// Mitsubishi GX Works2 project: 4LightsSeqLDv2   PLC: FX2N/FX2NC
// Examples Algorithm of 4 Lights on in seq then off in seq

// global labels: Global1
VAR_GLOBAL
  Step1 AT S10 : BOOL;  (* Inital Step *)
  Step2 AT S11 : BOOL;
  Step3 AT S12 : BOOL;
  Step4 AT S13 : BOOL;
  Step5 AT S14 : BOOL;
  Step6 AT S15 : BOOL;
  Step7 AT S16 : BOOL;
  Step8 AT S17 : BOOL;
  Step9 AT S18 : BOOL;
  StartPB AT X000 : BOOL;  (* NO Momentary PB *)
  StopPB AT X001 : BOOL;  (* NC Momentary PB *)
  PL1 AT Y000 : BOOL;
  PL2 AT Y001 : BOOL;
  PL3 AT Y002 : BOOL;
  PL4 AT Y003 : BOOL;
  SC : BOOL;  (* State Changed *)
  CurrentState AT D100 : WORD;
  PreviousState AT D101 : WORD;
  S1ToS2 : BOOL;
  S2ToS3 : BOOL;
  S3ToS4 : BOOL;
  S4ToS5 : BOOL;
  S5ToS6 : BOOL;
  S6ToS7 : BOOL;
  S7ToS8 : BOOL;
  S8ToS9 : BOOL;
  S9ToS1 : BOOL;
  Do_Shift : BOOL;
  Src_Bit : BOOL;
  First_Start : BOOL;
  Step0 AT S9 : BOOL;
  StepCtr : CTU;
  Stp_Ary : ARRAY [0..15] OF BOOL;
  Stp_Idx : INT;
  StpDn_Ary : ARRAY [0..15] OF BOOL;
  Get_Step_1 : Get_Step;
  Do_Count : BOOL;
  Stp_Ary_D : ARRAY [0..15] OF BOOL;
  StpDn_Ary_D : ARRAY [0..15] OF BOOL;
END_VAR

// task Task_01 (event TRUE, interval 0, priority 31): FSM_DRUM

PROGRAM FSM_SR_NO_SC
(* structured ladder/FBD written out as ST: instructions are called as NAME(EN, inputs, outputs); _pN, _eN, _tN stand for wires *)
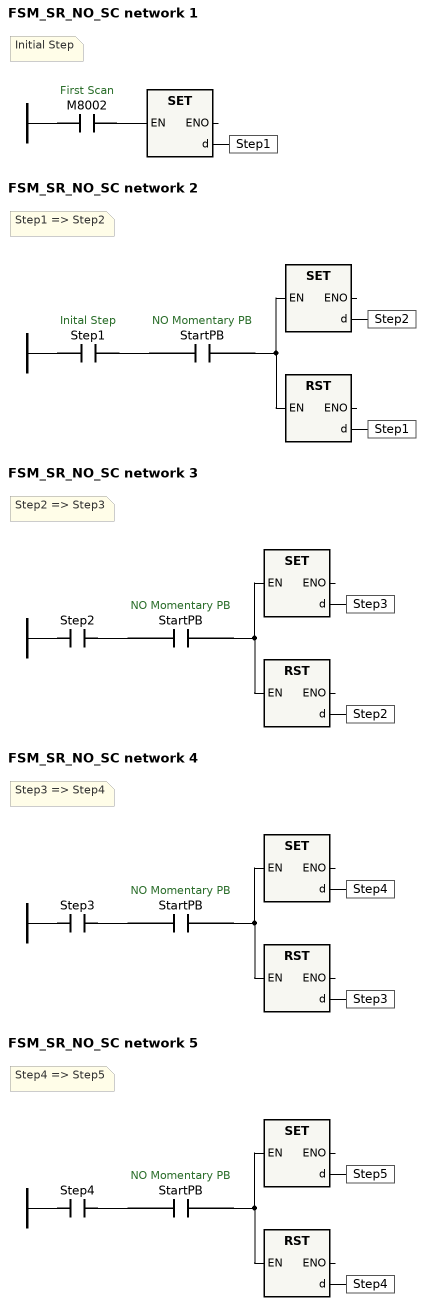
(* network 1 *)
(* Initial Step *)
SET(M8002, Step1);
(* network 2 *)
(* Step1 => Step2 *)
_p1 := Step1 AND StartPB;
SET(_p1, Step2);
RST(_p1, Step1);
(* network 3 *)
(* Step2 => Step3 *)
_p1 := Step2 AND StartPB;
SET(_p1, Step3);
RST(_p1, Step2);
(* network 4 *)
(* Step3 => Step4 *)
_p1 := Step3 AND StartPB;
SET(_p1, Step4);
RST(_p1, Step3);
(* network 5 *)
(* Step4 => Step5 *)
_p1 := Step4 AND StartPB;
SET(_p1, Step5);
RST(_p1, Step4);
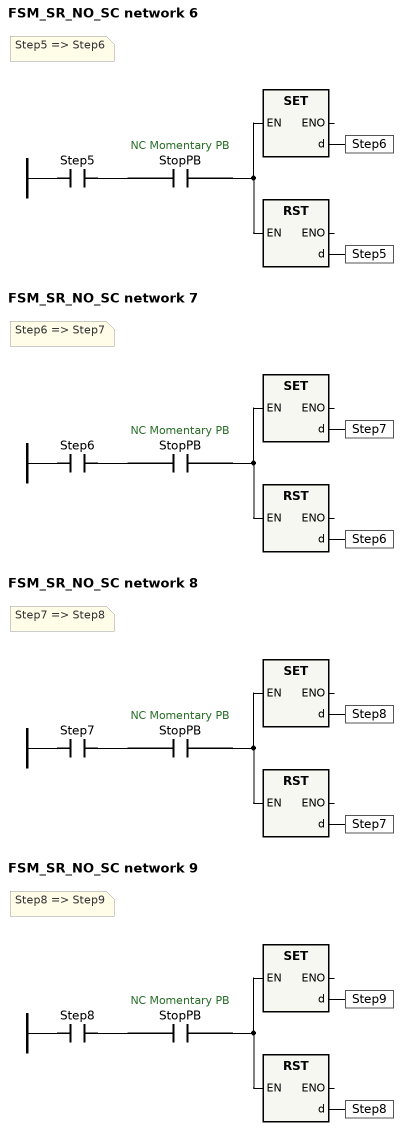
(* network 6 *)
(* Step5 => Step6 *)
_p1 := Step5 AND StopPB;
SET(_p1, Step6);
RST(_p1, Step5);
(* network 7 *)
(* Step6 => Step7 *)
_p1 := Step6 AND StopPB;
SET(_p1, Step7);
RST(_p1, Step6);
(* network 8 *)
(* Step7 => Step8 *)
_p1 := Step7 AND StopPB;
SET(_p1, Step8);
RST(_p1, Step7);
(* network 9 *)
(* Step8 => Step9 *)
_p1 := Step8 AND StopPB;
SET(_p1, Step9);
RST(_p1, Step8);
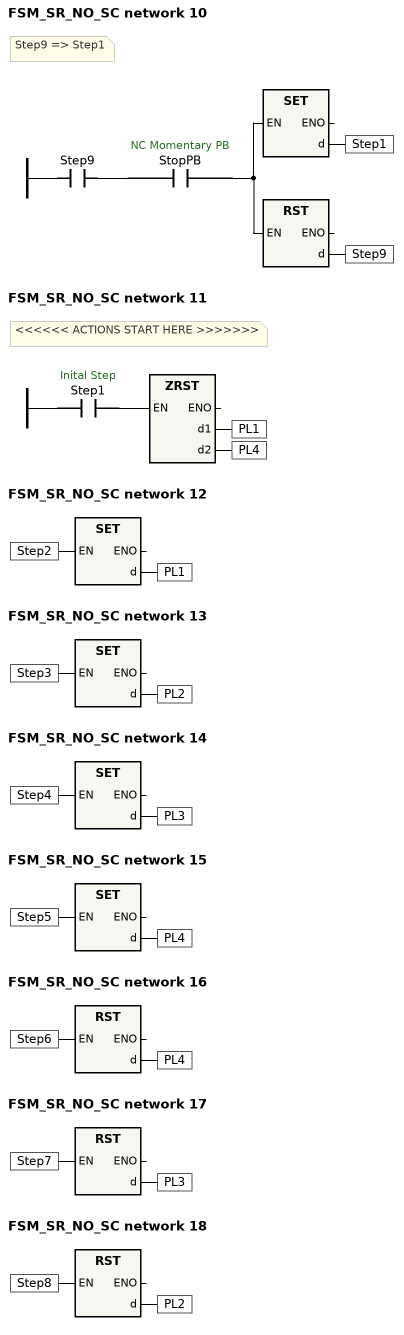
(* network 10 *)
(* Step9 => Step1 *)
_p1 := Step9 AND StopPB;
SET(_p1, Step1);
RST(_p1, Step9);
(* network 11 *)
(* <<<<<< ACTIONS START HERE >>>>>>> *)
ZRST(Step1, PL1, PL4);
(* network 12 *)
SET(Step2, PL1);
(* network 13 *)
SET(Step3, PL2);
(* network 14 *)
SET(Step4, PL3);
(* network 15 *)
SET(Step5, PL4);
(* network 16 *)
RST(Step6, PL4);
(* network 17 *)
RST(Step7, PL3);
(* network 18 *)
RST(Step8, PL2);
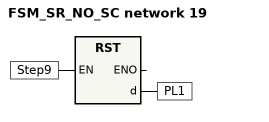
(* network 19 *)
RST(Step9, PL1);
END_PROGRAM

PROGRAM FSM_SR_SC
(* structured ladder/FBD written out as ST: instructions are called as NAME(EN, inputs, outputs); _pN, _eN, _tN stand for wires *)
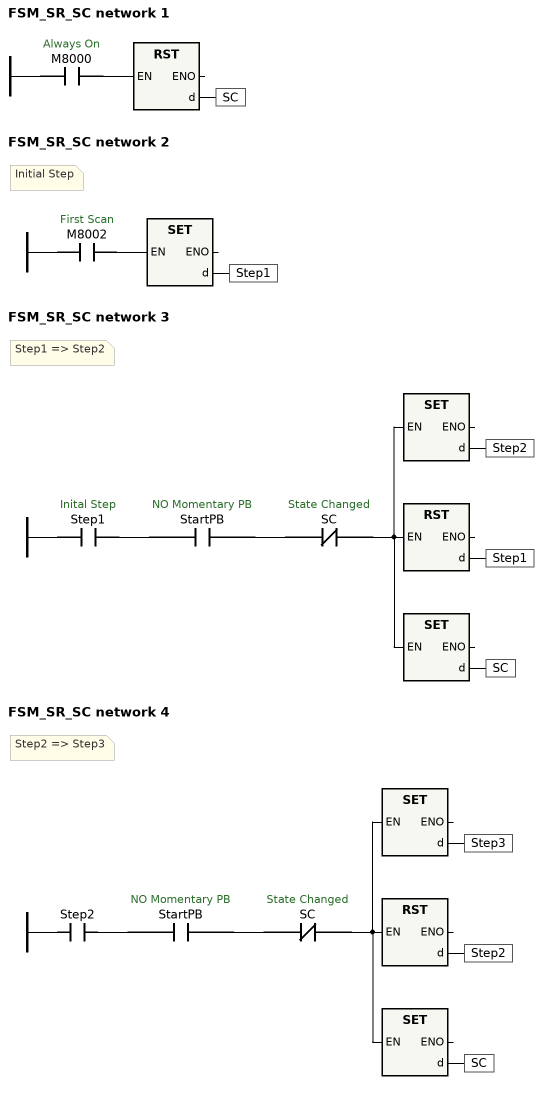
(* network 1 *)
RST(M8000, SC);
(* network 2 *)
(* Initial Step *)
SET(M8002, Step1);
(* network 3 *)
(* Step1 => Step2 *)
_p1 := Step1 AND StartPB AND NOT SC;
SET(_p1, Step2);
RST(_p1, Step1);
SET(_p1, SC);
(* network 4 *)
(* Step2 => Step3 *)
_p1 := Step2 AND StartPB AND NOT SC;
SET(_p1, Step3);
RST(_p1, Step2);
SET(_p1, SC);
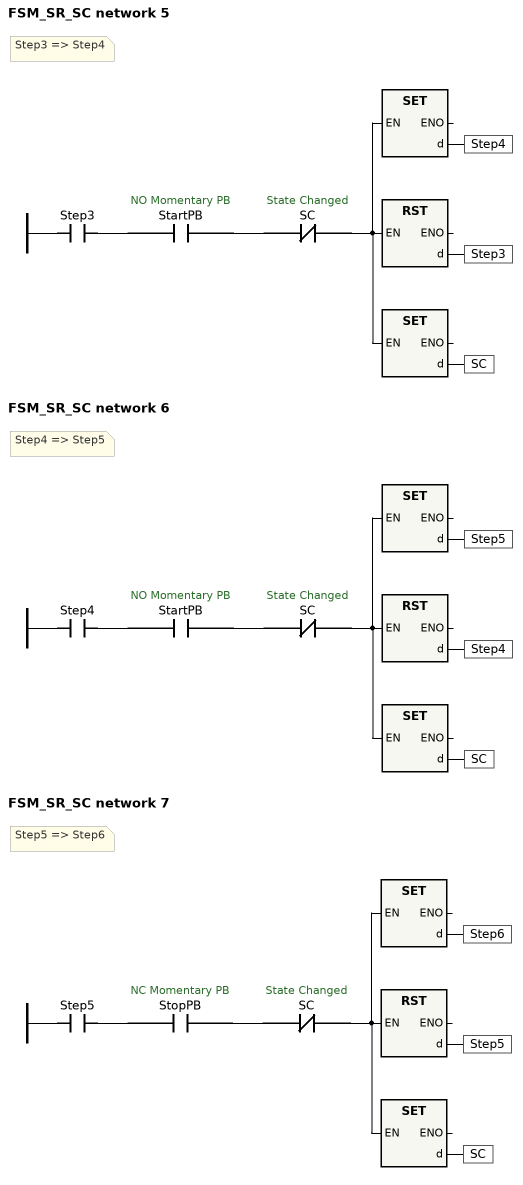
(* network 5 *)
(* Step3 => Step4 *)
_p1 := Step3 AND StartPB AND NOT SC;
SET(_p1, Step4);
RST(_p1, Step3);
SET(_p1, SC);
(* network 6 *)
(* Step4 => Step5 *)
_p1 := Step4 AND StartPB AND NOT SC;
SET(_p1, Step5);
RST(_p1, Step4);
SET(_p1, SC);
(* network 7 *)
(* Step5 => Step6 *)
_p1 := Step5 AND StopPB AND NOT SC;
SET(_p1, Step6);
RST(_p1, Step5);
SET(_p1, SC);
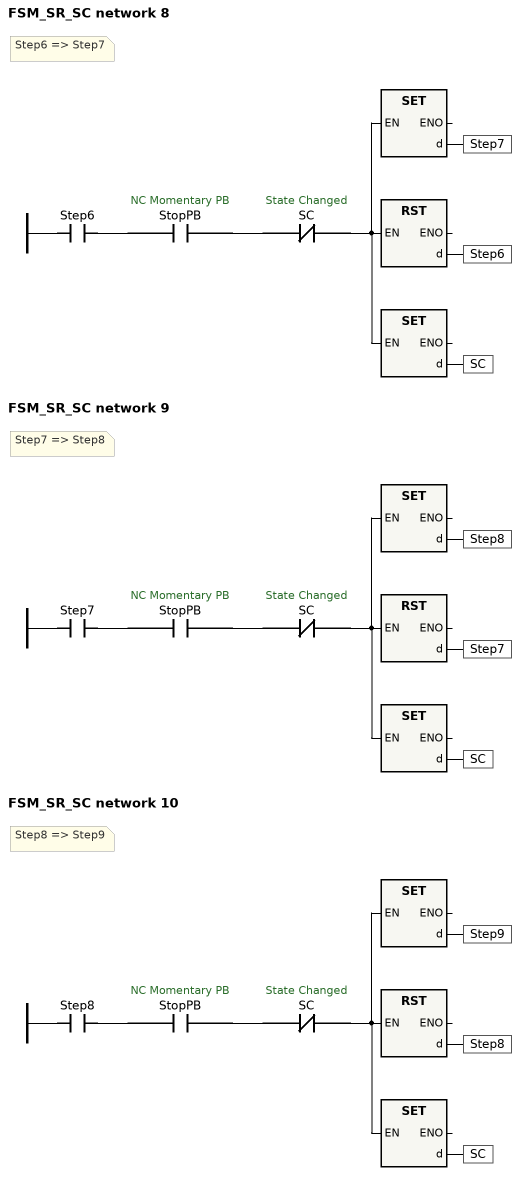
(* network 8 *)
(* Step6 => Step7 *)
_p1 := Step6 AND StopPB AND NOT SC;
SET(_p1, Step7);
RST(_p1, Step6);
SET(_p1, SC);
(* network 9 *)
(* Step7 => Step8 *)
_p1 := Step7 AND StopPB AND NOT SC;
SET(_p1, Step8);
RST(_p1, Step7);
SET(_p1, SC);
(* network 10 *)
(* Step8 => Step9 *)
_p1 := Step8 AND StopPB AND NOT SC;
SET(_p1, Step9);
RST(_p1, Step8);
SET(_p1, SC);
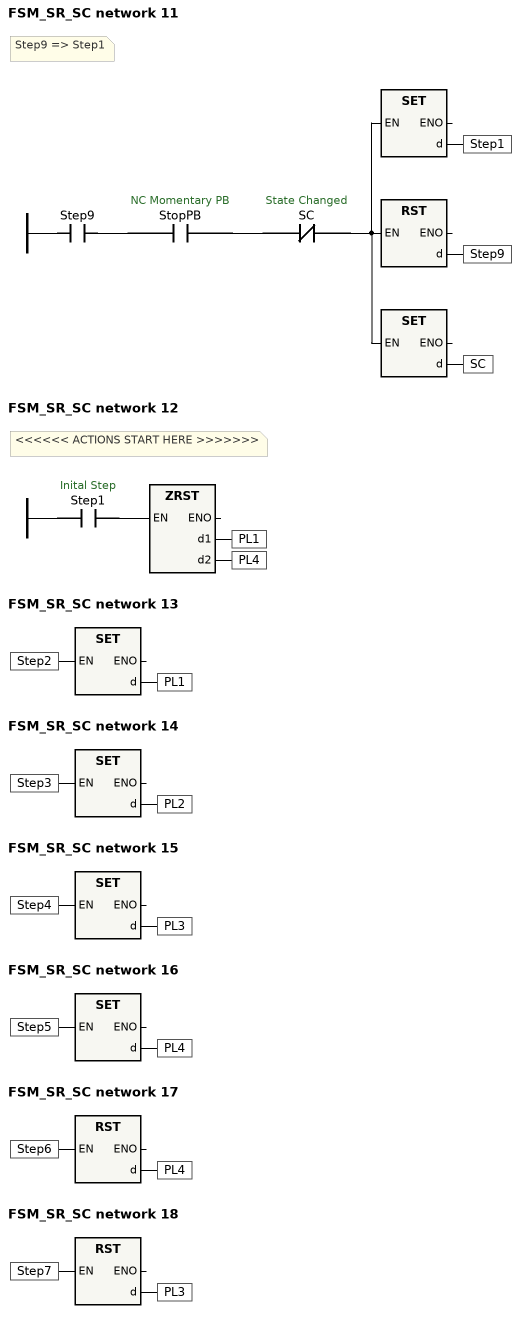
(* network 11 *)
(* Step9 => Step1 *)
_p1 := Step9 AND StopPB AND NOT SC;
SET(_p1, Step1);
RST(_p1, Step9);
SET(_p1, SC);
(* network 12 *)
(* <<<<<< ACTIONS START HERE >>>>>>> *)
ZRST(Step1, PL1, PL4);
(* network 13 *)
SET(Step2, PL1);
(* network 14 *)
SET(Step3, PL2);
(* network 15 *)
SET(Step4, PL3);
(* network 16 *)
SET(Step5, PL4);
(* network 17 *)
RST(Step6, PL4);
(* network 18 *)
RST(Step7, PL3);
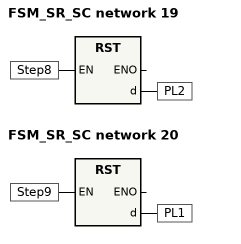
(* network 19 *)
RST(Step8, PL2);
(* network 20 *)
RST(Step9, PL1);
END_PROGRAM

PROGRAM FSM_EQU
(* structured ladder/FBD written out as ST: instructions are called as NAME(EN, inputs, outputs); _pN, _eN, _tN stand for wires *)
(* Instructions Supported in Simulator and LE3U Trainer *)
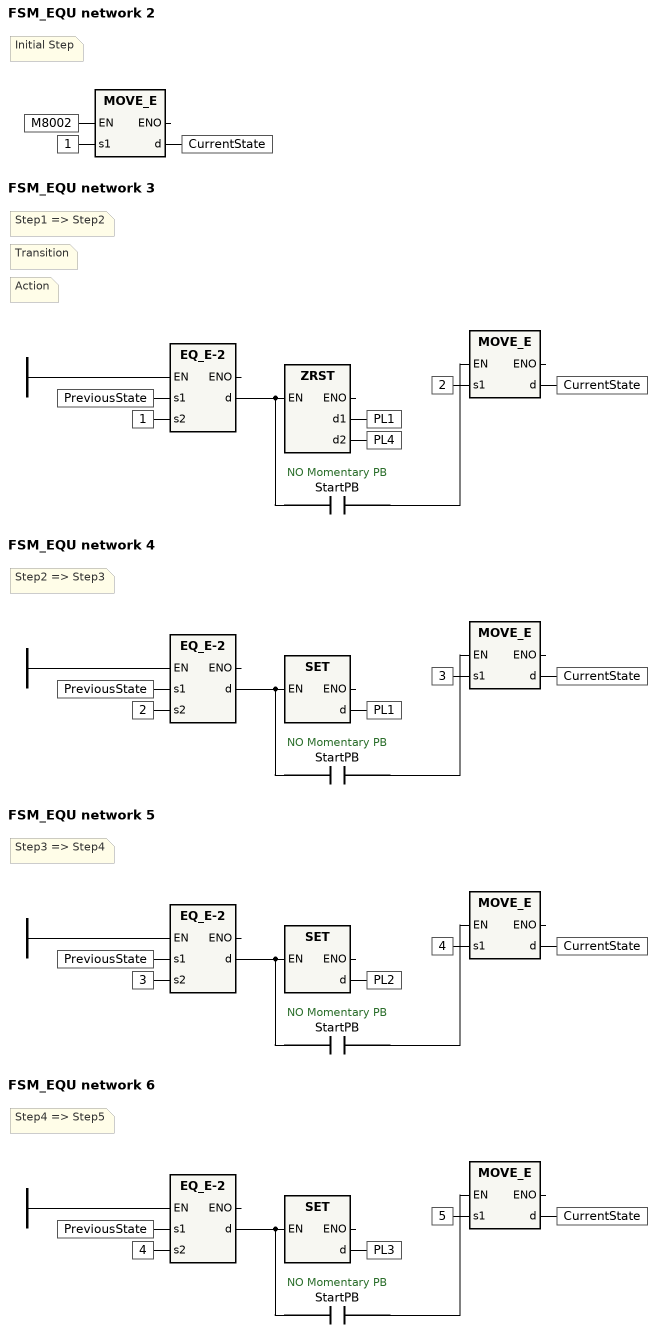
(* network 2 *)
(* Initial Step *)
MOVE_E(M8002, 1, CurrentState);
(* network 3 *)
(* Step1 => Step2 *)
(* Transition *)
(* Action *)
EQ_E(TRUE, PreviousState, 1, _t1);
MOVE_E(_t1 AND StartPB, 2, CurrentState);
ZRST(_t1, PL1, PL4);
(* network 4 *)
(* Step2 => Step3 *)
EQ_E(TRUE, PreviousState, 2, _t1);
MOVE_E(_t1 AND StartPB, 3, CurrentState);
SET(_t1, PL1);
(* network 5 *)
(* Step3 => Step4 *)
EQ_E(TRUE, PreviousState, 3, _t1);
MOVE_E(_t1 AND StartPB, 4, CurrentState);
SET(_t1, PL2);
(* network 6 *)
(* Step4 => Step5 *)
EQ_E(TRUE, PreviousState, 4, _t1);
MOVE_E(_t1 AND StartPB, 5, CurrentState);
SET(_t1, PL3);
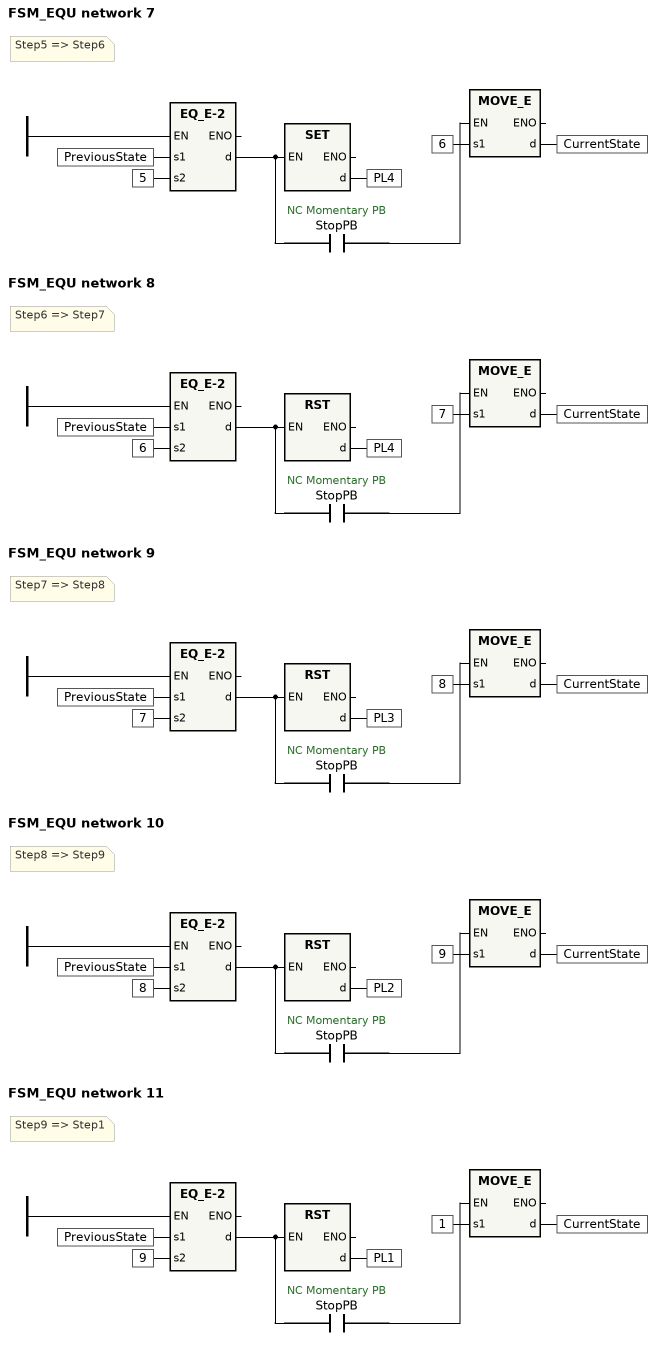
(* network 7 *)
(* Step5 => Step6 *)
EQ_E(TRUE, PreviousState, 5, _t1);
MOVE_E(_t1 AND StopPB, 6, CurrentState);
SET(_t1, PL4);
(* network 8 *)
(* Step6 => Step7 *)
EQ_E(TRUE, PreviousState, 6, _t1);
MOVE_E(_t1 AND StopPB, 7, CurrentState);
RST(_t1, PL4);
(* network 9 *)
(* Step7 => Step8 *)
EQ_E(TRUE, PreviousState, 7, _t1);
MOVE_E(_t1 AND StopPB, 8, CurrentState);
RST(_t1, PL3);
(* network 10 *)
(* Step8 => Step9 *)
EQ_E(TRUE, PreviousState, 8, _t1);
MOVE_E(_t1 AND StopPB, 9, CurrentState);
RST(_t1, PL2);
(* network 11 *)
(* Step9 => Step1 *)
EQ_E(TRUE, PreviousState, 9, _t1);
MOVE_E(_t1 AND StopPB, 1, CurrentState);
RST(_t1, PL1);
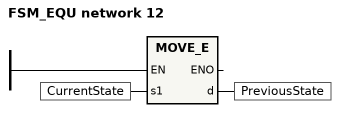
(* network 12 *)
MOVE_E(TRUE, CurrentState, PreviousState);
END_PROGRAM

PROGRAM FSM_PN
(* structured ladder/FBD written out as ST: instructions are called as NAME(EN, inputs, outputs); _pN, _eN, _tN stand for wires *)
(* Finite State Machine / Using Petri Net Techique *)
(* Transitions *)
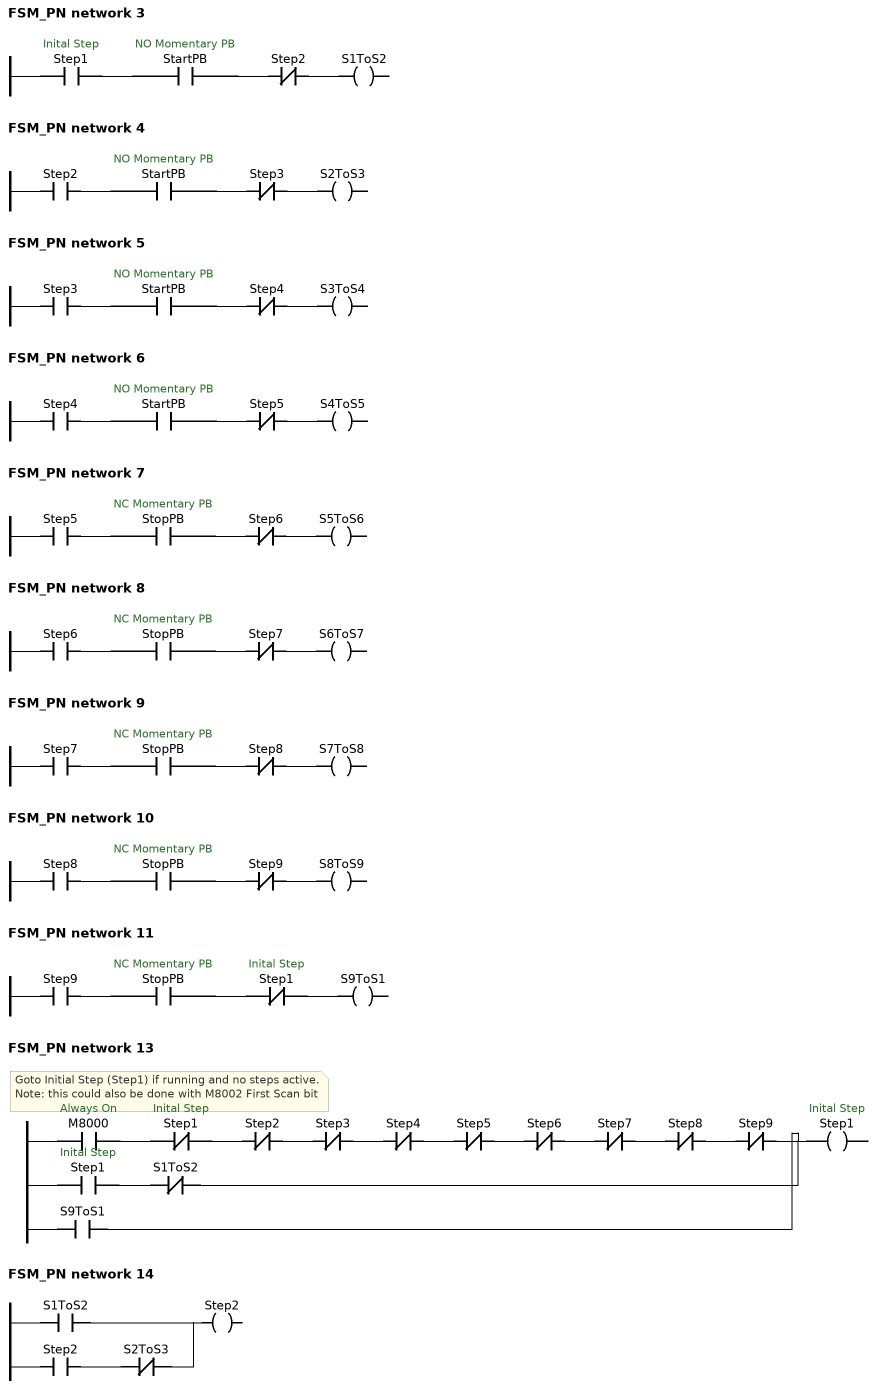
(* network 3 *)
S1ToS2 := Step1 AND StartPB AND NOT Step2;
(* network 4 *)
S2ToS3 := Step2 AND StartPB AND NOT Step3;
(* network 5 *)
S3ToS4 := Step3 AND StartPB AND NOT Step4;
(* network 6 *)
S4ToS5 := Step4 AND StartPB AND NOT Step5;
(* network 7 *)
S5ToS6 := Step5 AND StopPB AND NOT Step6;
(* network 8 *)
S6ToS7 := Step6 AND StopPB AND NOT Step7;
(* network 9 *)
S7ToS8 := Step7 AND StopPB AND NOT Step8;
(* network 10 *)
S8ToS9 := Step8 AND StopPB AND NOT Step9;
(* network 11 *)
S9ToS1 := Step9 AND StopPB AND NOT Step1;
(* Step Logic *)
(* network 13 *)
(* Goto Initial Step (Step1) if running and no steps active. Note: this could also be done with M8002 First Scan bit *)
Step1 := (M8000 AND NOT Step1 AND NOT Step2 AND NOT Step3 AND NOT Step4 AND NOT Step5 AND NOT Step6 AND NOT Step7 AND NOT Step8 AND NOT Step9) OR (Step1 AND NOT S1ToS2) OR S9ToS1;
(* network 14 *)
Step2 := S1ToS2 OR (Step2 AND NOT S2ToS3);
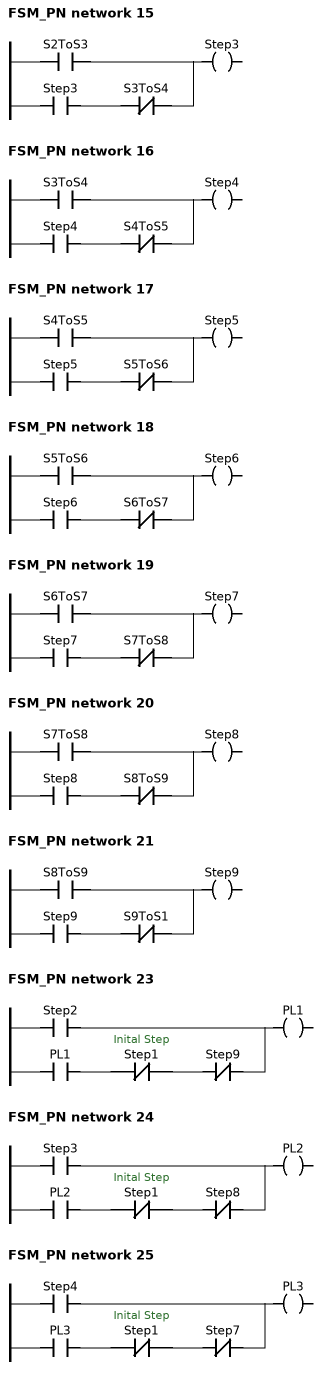
(* network 15 *)
Step3 := S2ToS3 OR (Step3 AND NOT S3ToS4);
(* network 16 *)
Step4 := S3ToS4 OR (Step4 AND NOT S4ToS5);
(* network 17 *)
Step5 := S4ToS5 OR (Step5 AND NOT S5ToS6);
(* network 18 *)
Step6 := S5ToS6 OR (Step6 AND NOT S6ToS7);
(* network 19 *)
Step7 := S6ToS7 OR (Step7 AND NOT S7ToS8);
(* network 20 *)
Step8 := S7ToS8 OR (Step8 AND NOT S8ToS9);
(* network 21 *)
Step9 := S8ToS9 OR (Step9 AND NOT S9ToS1);
(* Actions *)
(* network 23 *)
PL1 := Step2 OR (PL1 AND NOT Step1 AND NOT Step9);
(* network 24 *)
PL2 := Step3 OR (PL2 AND NOT Step1 AND NOT Step8);
(* network 25 *)
PL3 := Step4 OR (PL3 AND NOT Step1 AND NOT Step7);
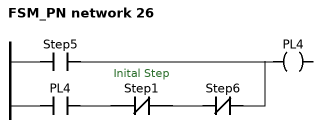
(* network 26 *)
PL4 := Step5 OR (PL4 AND NOT Step1 AND NOT Step6);
END_PROGRAM

PROGRAM FSM_SHL
(* structured ladder/FBD written out as ST: instructions are called as NAME(EN, inputs, outputs); _pN, _eN, _tN stand for wires *)
(* Finite State Machine / Using Shift Left *)
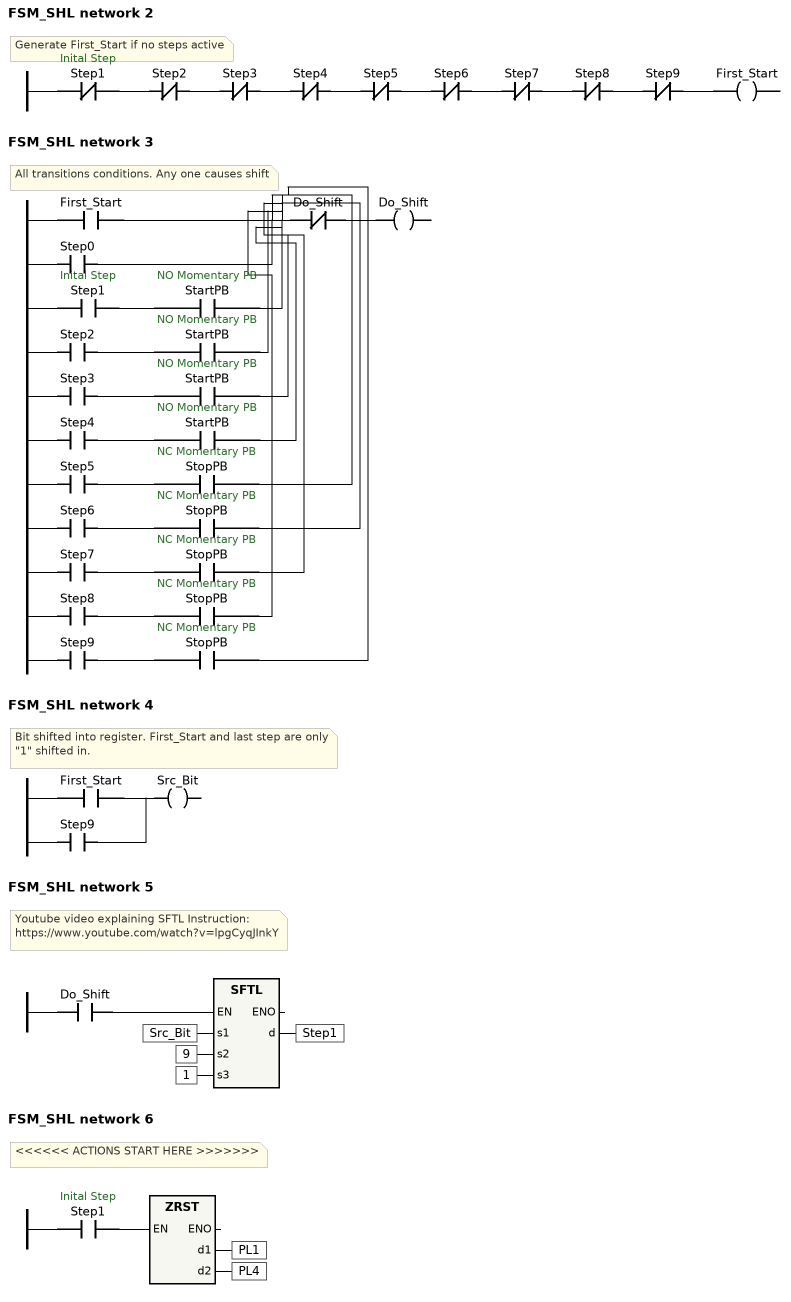
(* network 2 *)
(* Generate First_Start if no steps active *)
First_Start := NOT Step1 AND NOT Step2 AND NOT Step3 AND NOT Step4 AND NOT Step5 AND NOT Step6 AND NOT Step7 AND NOT Step8 AND NOT Step9;
(* network 3 *)
(* All transitions conditions. Any one causes shift *)
Do_Shift := (First_Start OR Step0 OR (Step1 AND StartPB) OR (Step2 AND StartPB) OR (Step3 AND StartPB) OR (Step4 AND StartPB) OR (Step5 AND StopPB) OR (Step6 AND StopPB) OR (Step7 AND StopPB) OR (Step8 AND StopPB) OR (Step9 AND StopPB)) AND NOT Do_Shift;
(* network 4 *)
(* Bit shifted into register. First_Start and last step are only "1" shifted in. *)
Src_Bit := First_Start OR Step9;
(* network 5 *)
(* Youtube video explaining SFTL Instruction: / https://www.youtube.com/watch?v=lpgCyqJInkY *)
SFTL(Do_Shift, Src_Bit, 9, 1, Step1);
(* network 6 *)
(* <<<<<< ACTIONS START HERE >>>>>>> *)
ZRST(Step1, PL1, PL4);
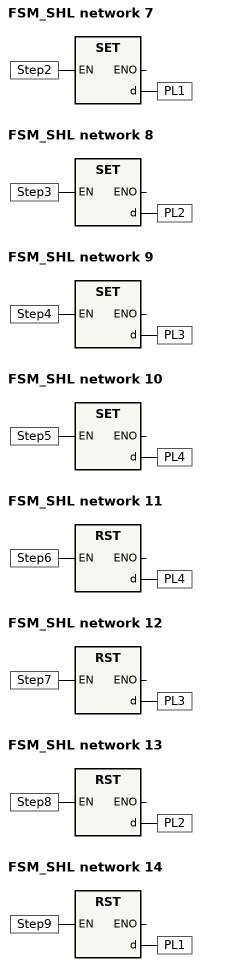
(* network 7 *)
SET(Step2, PL1);
(* network 8 *)
SET(Step3, PL2);
(* network 9 *)
SET(Step4, PL3);
(* network 10 *)
SET(Step5, PL4);
(* network 11 *)
RST(Step6, PL4);
(* network 12 *)
RST(Step7, PL3);
(* network 13 *)
RST(Step8, PL2);
(* network 14 *)
RST(Step9, PL1);
END_PROGRAM

PROGRAM FSM_STL
(* structured ladder/FBD written out as ST: instructions are called as NAME(EN, inputs, outputs); _pN, _eN, _tN stand for wires *)
(* Instructions Supported in Simulator and LE3U Trainer *)
(* STL - Stands for Step Ladder. Be aware that Siemens PLC have a "STL" which stands for Statement List which is essentially Instruction List (IL). /  / A lot of Asian made PLCs have STL (Step Ladder) but only one USA PLC has anything like it. Domore has Stage Programming which is very similiar to STL and you will do a lab using Stage Programming. *)
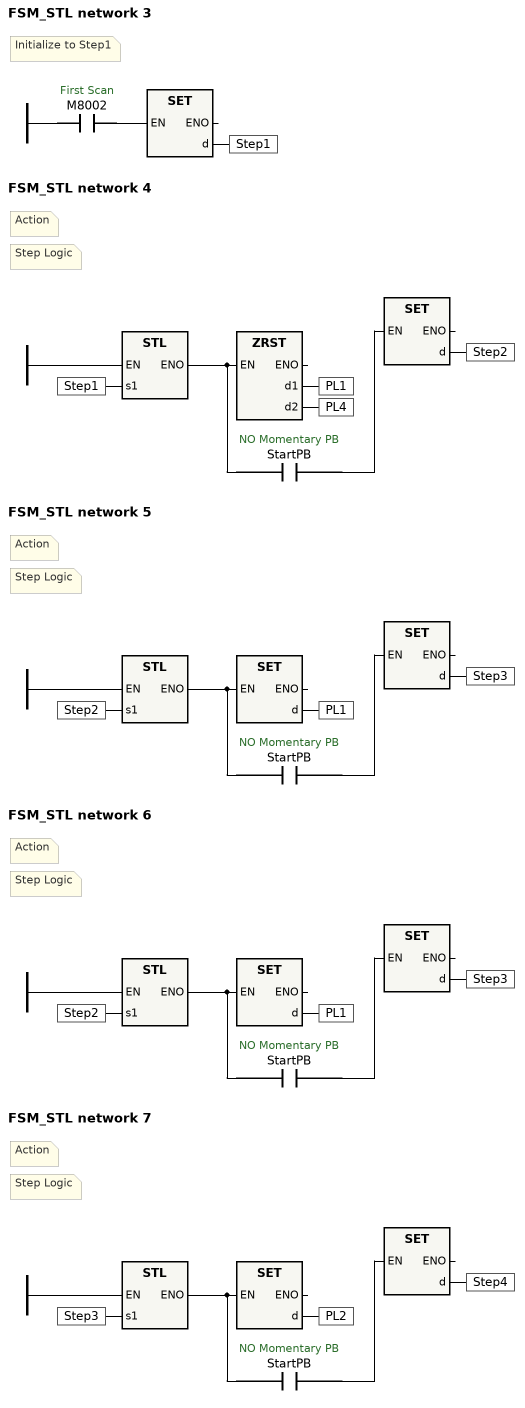
(* network 3 *)
(* Initialize to Step1 *)
SET(M8002, Step1);
(* network 4 *)
(* Action *)
(* Step Logic *)
_e1 := STL(TRUE, Step1);
ZRST(_e1, PL1, PL4);
SET(_e1 AND StartPB, Step2);
(* network 5 *)
(* Action *)
(* Step Logic *)
_e1 := STL(TRUE, Step2);
SET(_e1, PL1);
SET(_e1 AND StartPB, Step3);
(* network 6 *)
(* Action *)
(* Step Logic *)
_e1 := STL(TRUE, Step2);
SET(_e1, PL1);
SET(_e1 AND StartPB, Step3);
(* network 7 *)
(* Action *)
(* Step Logic *)
_e1 := STL(TRUE, Step3);
SET(_e1, PL2);
SET(_e1 AND StartPB, Step4);
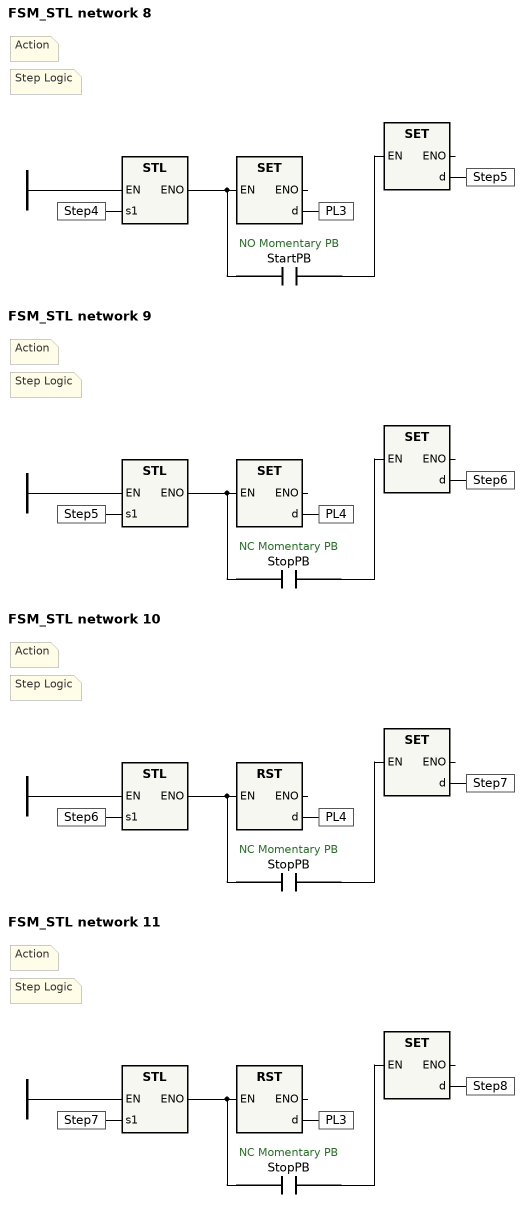
(* network 8 *)
(* Action *)
(* Step Logic *)
_e1 := STL(TRUE, Step4);
SET(_e1, PL3);
SET(_e1 AND StartPB, Step5);
(* network 9 *)
(* Action *)
(* Step Logic *)
_e1 := STL(TRUE, Step5);
SET(_e1, PL4);
SET(_e1 AND StopPB, Step6);
(* network 10 *)
(* Action *)
(* Step Logic *)
_e1 := STL(TRUE, Step6);
RST(_e1, PL4);
SET(_e1 AND StopPB, Step7);
(* network 11 *)
(* Action *)
(* Step Logic *)
_e1 := STL(TRUE, Step7);
RST(_e1, PL3);
SET(_e1 AND StopPB, Step8);
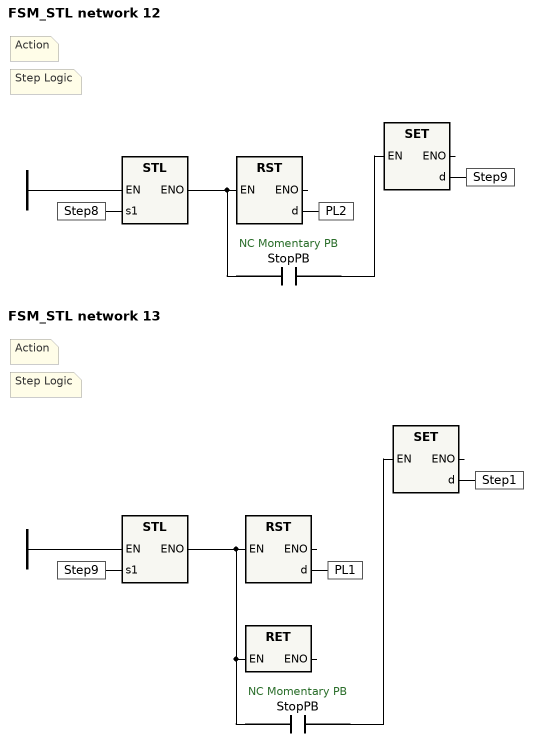
(* network 12 *)
(* Action *)
(* Step Logic *)
_e1 := STL(TRUE, Step8);
RST(_e1, PL2);
SET(_e1 AND StopPB, Step9);
(* network 13 *)
(* Action *)
(* Step Logic *)
_e1 := STL(TRUE, Step9);
RST(_e1, PL1);
SET(_e1 AND StopPB, Step1);
RET(_e1);
END_PROGRAM

FUNCTION_BLOCK Get_Step
VAR_OUTPUT
  GSOut : BOOL;
END_VAR
VAR_IN_OUT
  SArray : ARRAY [0..15] OF BOOL;
END_VAR
VAR_INPUT
  StpNum : INT;
END_VAR
GSOut := SArray[StpNum];
END_FUNCTION_BLOCK

FUNCTION_BLOCK SR_Step
VAR_INPUT
  In : BOOL;
  StpNum : INT;
END_VAR
VAR_IN_OUT
  SArray : ARRAY [0..15] OF BOOL;
END_VAR
SArray[StpNum] := In;
END_FUNCTION_BLOCK

PROGRAM FSM_DRUM
(* structured ladder/FBD written out as ST: instructions are called as NAME(EN, inputs, outputs); _pN, _eN, _tN stand for wires *)
(* Instructions Supported in Simulator and LE3U Trainer /  / Requires Initalize POU to be running also. *)
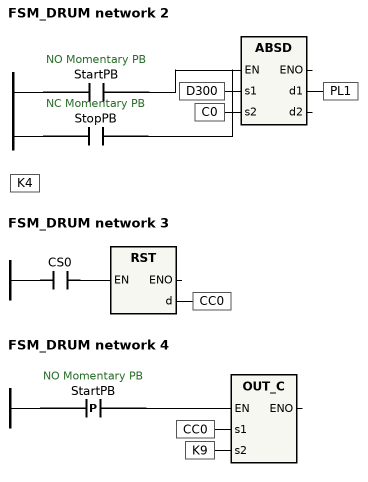
(* network 2 *)
ABSD(StartPB OR StopPB, D300, C0, PL1, _open);
(* not connected to any output: K4 *)
(* network 3 *)
RST(CS0, CC0);
(* network 4 *)
OUT_C(LDP(TRUE, StartPB), CC0, K9);
END_PROGRAM

PROGRAM Initialize
D300 := 2;
D301 := 9;
D302 := 3;
D303 := 8;
D304 := 4;
D305 := 7;
D306 := 5;
D307 := 6;
END_PROGRAM

PROGRAM FSM_Counter_Decode
(* structured ladder/FBD written out as ST: instructions are called as NAME(EN, inputs, outputs); _pN, _eN, _tN stand for wires *)
(* Instructions Supported in Simulator Only. Instruction DEC not supported in LE3U Trainer *)
(* Finite State Machine / Using Counter and Decode Instructions. *)
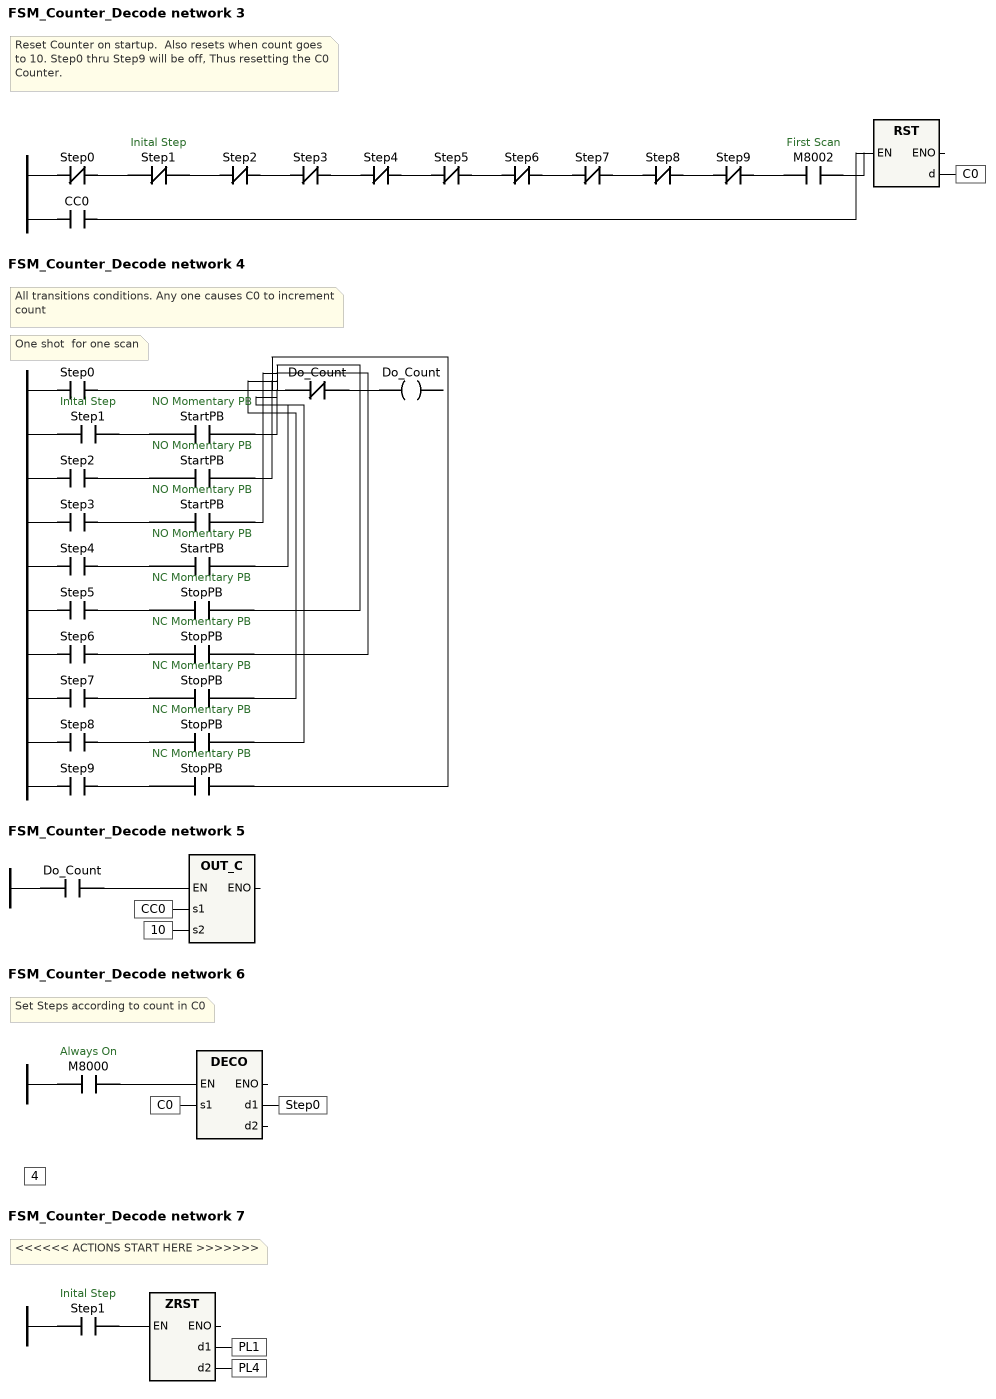
(* network 3 *)
(* Reset Counter on startup.  Also resets when count goes to 10. Step0 thru Step9 will be off, Thus resetting the C0 Counter. *)
RST((NOT Step0 AND NOT Step1 AND NOT Step2 AND NOT Step3 AND NOT Step4 AND NOT Step5 AND NOT Step6 AND NOT Step7 AND NOT Step8 AND NOT Step9 AND M8002) OR CC0, C0);
(* network 4 *)
(* All transitions conditions. Any one causes C0 to increment count *)
(* One shot  for one scan *)
Do_Count := (Step0 OR (Step1 AND StartPB) OR (Step2 AND StartPB) OR (Step3 AND StartPB) OR (Step4 AND StartPB) OR (Step5 AND StopPB) OR (Step6 AND StopPB) OR (Step7 AND StopPB) OR (Step8 AND StopPB) OR (Step9 AND StopPB)) AND NOT Do_Count;
(* network 5 *)
OUT_C(Do_Count, CC0, 10);
(* network 6 *)
(* Set Steps according to count in C0 *)
DECO(M8000, C0, Step0, _open);
(* not connected to any output: 4 *)
(* network 7 *)
(* <<<<<< ACTIONS START HERE >>>>>>> *)
ZRST(Step1, PL1, PL4);
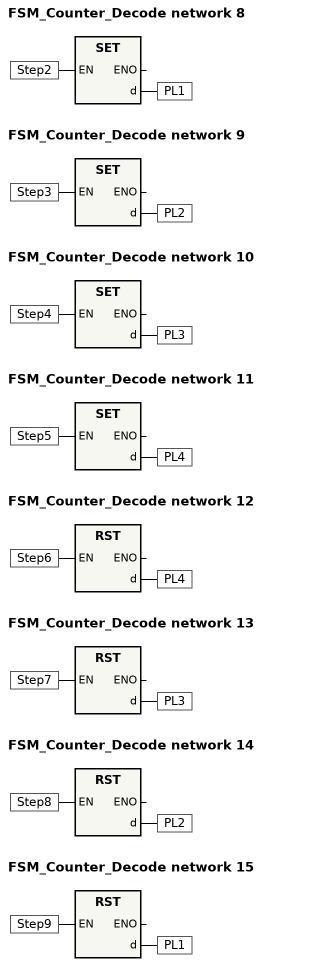
(* network 8 *)
SET(Step2, PL1);
(* network 9 *)
SET(Step3, PL2);
(* network 10 *)
SET(Step4, PL3);
(* network 11 *)
SET(Step5, PL4);
(* network 12 *)
RST(Step6, PL4);
(* network 13 *)
RST(Step7, PL3);
(* network 14 *)
RST(Step8, PL2);
(* network 15 *)
RST(Step9, PL1);
END_PROGRAM

PROGRAM FSM_Counter
VAR
  StepCtrCV : INT;
  ClrStep : SR_Step;
  SetStep : SR_Step;
  Reset : BOOL;
  Do_Jump : BOOL;
  Step_Jump : INT;
  R_TRIG_1 : R_TRIG;
END_VAR
(* structured ladder/FBD written out as ST: instructions are called as NAME(EN, inputs, outputs); _pN, _eN, _tN stand for wires *)
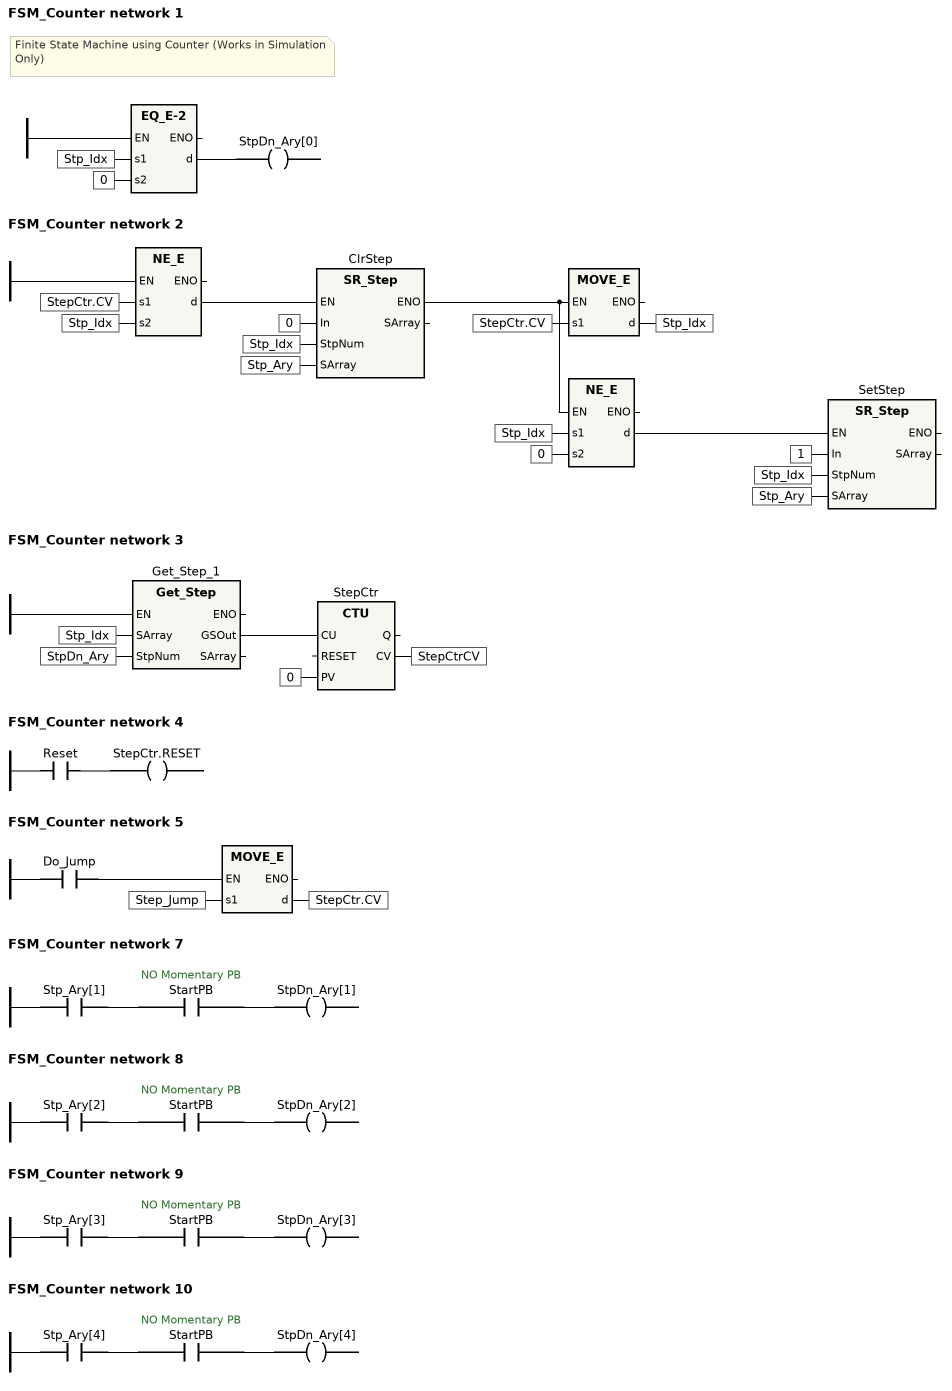
(* network 1 *)
(* Finite State Machine using Counter (Works in Simulation Only) *)
EQ_E(TRUE, Stp_Idx, 0, _t1);
StpDn_Ary[0] := _t1;
(* network 2 *)
NE_E(TRUE, StepCtr.CV, Stp_Idx, _t1);
ClrStep(EN := _t1, In := 0, StpNum := Stp_Idx, SArray := Stp_Ary);
MOVE_E(ClrStep.ENO, StepCtr.CV, Stp_Idx);
NE_E(ClrStep.ENO, Stp_Idx, 0, _t2);
SetStep(EN := _t2, In := 1, StpNum := Stp_Idx, SArray := Stp_Ary);
(* network 3 *)
Get_Step_1(EN := TRUE, SArray := Stp_Idx, StpNum := StpDn_Ary);
StepCtr(CU := Get_Step_1.GSOut, PV := 0, CV => StepCtrCV);
(* network 4 *)
StepCtr.RESET := Reset;
(* network 5 *)
MOVE_E(Do_Jump, Step_Jump, StepCtr.CV);
(* Transition Logic *)
(* network 7 *)
StpDn_Ary[1] := Stp_Ary[1] AND StartPB;
(* network 8 *)
StpDn_Ary[2] := Stp_Ary[2] AND StartPB;
(* network 9 *)
StpDn_Ary[3] := Stp_Ary[3] AND StartPB;
(* network 10 *)
StpDn_Ary[4] := Stp_Ary[4] AND StartPB;
